{attribute 'Tc2GvlVarNames'}
VAR_GLOBAL
	
	upperStackerUnload : BOOL;
	lowerStackerUnload : BOOL;
	upperStackerExternalCounterReset : BOOL;
	lowerStackerExternalCounterReset : BOOL;

END_VAR

(* stored: Version 1.1.0.1
   GVL GVL_InterConnection: Id {0fa15f22-3973-431f-9642-0bf4c5e6b236} *)
